FUNCTION_BLOCK LReal_To_Int (* Composite Function Block Type *)
  (* Standard: 61499-2 *)
  (* Version 0.0, 2012-01-01, 4DIAC-IDE, 4DIAC-Consortium *)
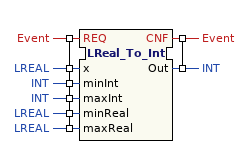
  EVENT_INPUT
    REQ WITH x, minInt, maxInt, minReal, maxReal; (* Normal Execution Request *)
  END_EVENT
  EVENT_OUTPUT
    CNF WITH Out; (* Execution Confirmation *)
  END_EVENT
  VAR_INPUT
    x : LREAL; (* Input event qualifier *)
    minInt : INT;
    maxInt : INT;
    minReal : LREAL;
    maxReal : LREAL;
  END_VAR
  VAR_OUTPUT
    Out : INT; (* Output event qualifier *)
  END_VAR
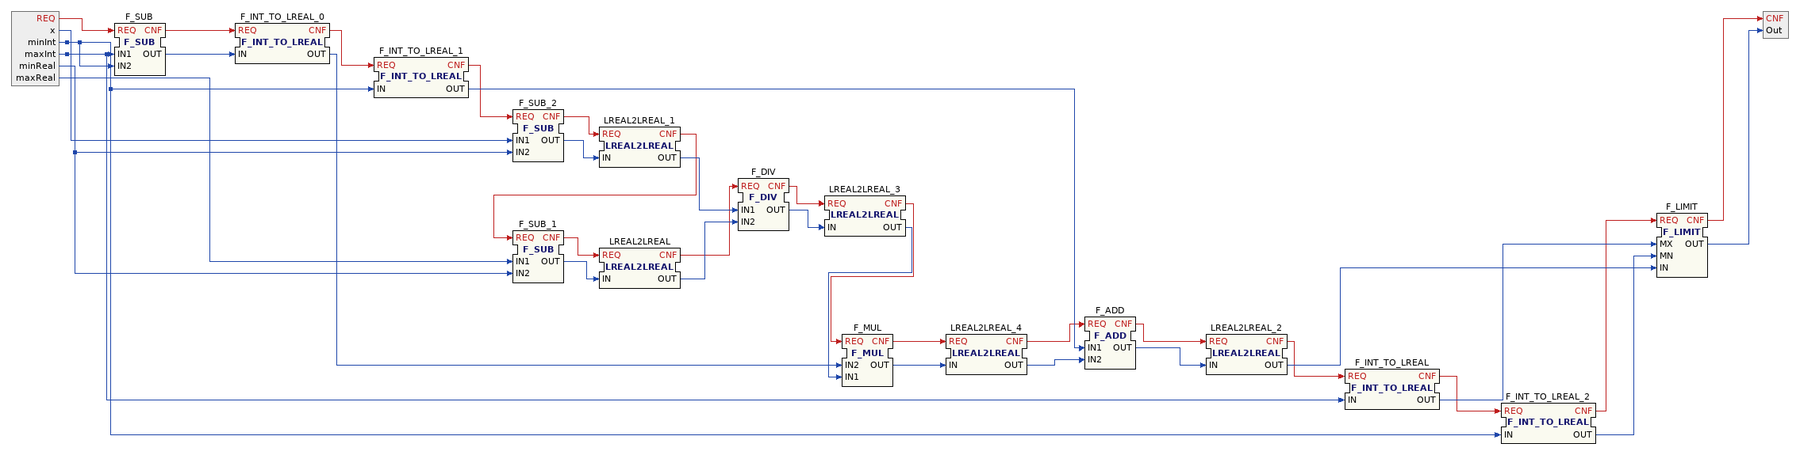
  FBS
    F_INT_TO_LREAL_0 : F_INT_TO_LREAL;
    F_INT_TO_LREAL_1 : F_INT_TO_LREAL;
    F_INT_TO_LREAL : F_INT_TO_LREAL;
    F_INT_TO_LREAL_2 : F_INT_TO_LREAL;
    F_LIMIT : F_LIMIT;
    F_SUB : F_SUB;
    F_SUB_1 : F_SUB;
    F_DIV : F_DIV;
    LREAL2LREAL : LREAL2LREAL;
    F_SUB_2 : F_SUB;
    LREAL2LREAL_1 : LREAL2LREAL;
    F_ADD : F_ADD;
    LREAL2LREAL_2 : LREAL2LREAL;
    F_MUL : F_MUL;
    LREAL2LREAL_3 : LREAL2LREAL;
    LREAL2LREAL_4 : LREAL2LREAL;
  END_FBS
  EVENT_CONNECTIONS
    F_INT_TO_LREAL_0.CNF TO F_INT_TO_LREAL_1.REQ;
    F_INT_TO_LREAL.CNF TO F_INT_TO_LREAL_2.REQ;
    REQ TO F_SUB.REQ;
    F_SUB.CNF TO F_INT_TO_LREAL_0.REQ;
    F_SUB_1.CNF TO LREAL2LREAL.REQ;
    F_INT_TO_LREAL_1.CNF TO F_SUB_2.REQ;
    F_SUB_2.CNF TO LREAL2LREAL_1.REQ;
    LREAL2LREAL_1.CNF TO F_SUB_1.REQ;
    LREAL2LREAL.CNF TO F_DIV.REQ;
    F_ADD.CNF TO LREAL2LREAL_2.REQ;
    F_DIV.CNF TO LREAL2LREAL_3.REQ;
    LREAL2LREAL_3.CNF TO F_MUL.REQ;
    F_MUL.CNF TO LREAL2LREAL_4.REQ;
    LREAL2LREAL_4.CNF TO F_ADD.REQ;
    LREAL2LREAL_2.CNF TO F_INT_TO_LREAL.REQ;
    F_LIMIT.CNF TO CNF;
    F_INT_TO_LREAL_2.CNF TO F_LIMIT.REQ;
  END_CONNECTIONS
  DATA_CONNECTIONS
    minInt TO F_INT_TO_LREAL_1.IN;
    minInt TO F_INT_TO_LREAL_2.IN;
    maxInt TO F_INT_TO_LREAL.IN;
    F_INT_TO_LREAL.OUT TO F_LIMIT.MX;
    F_INT_TO_LREAL_2.OUT TO F_LIMIT.MN;
    maxInt TO F_SUB.IN1;
    minInt TO F_SUB.IN2;
    F_SUB.OUT TO F_INT_TO_LREAL_0.IN;
    maxReal TO F_SUB_1.IN1;
    minReal TO F_SUB_1.IN2;
    F_SUB_1.OUT TO LREAL2LREAL.IN;
    x TO F_SUB_2.IN1;
    minReal TO F_SUB_2.IN2;
    F_SUB_2.OUT TO LREAL2LREAL_1.IN;
    LREAL2LREAL_1.OUT TO F_DIV.IN1;
    LREAL2LREAL.OUT TO F_DIV.IN2;
    F_INT_TO_LREAL_1.OUT TO F_ADD.IN1;
    LREAL2LREAL_2.OUT TO F_LIMIT.IN;
    F_ADD.OUT TO LREAL2LREAL_2.IN;
    F_INT_TO_LREAL_0.OUT TO F_MUL.IN2;
    F_DIV.OUT TO LREAL2LREAL_3.IN;
    LREAL2LREAL_3.OUT TO F_MUL.IN1;
    F_MUL.OUT TO LREAL2LREAL_4.IN;
    LREAL2LREAL_4.OUT TO F_ADD.IN2;
    F_LIMIT.OUT TO Out;
  END_CONNECTIONS
END_FUNCTION_BLOCK
